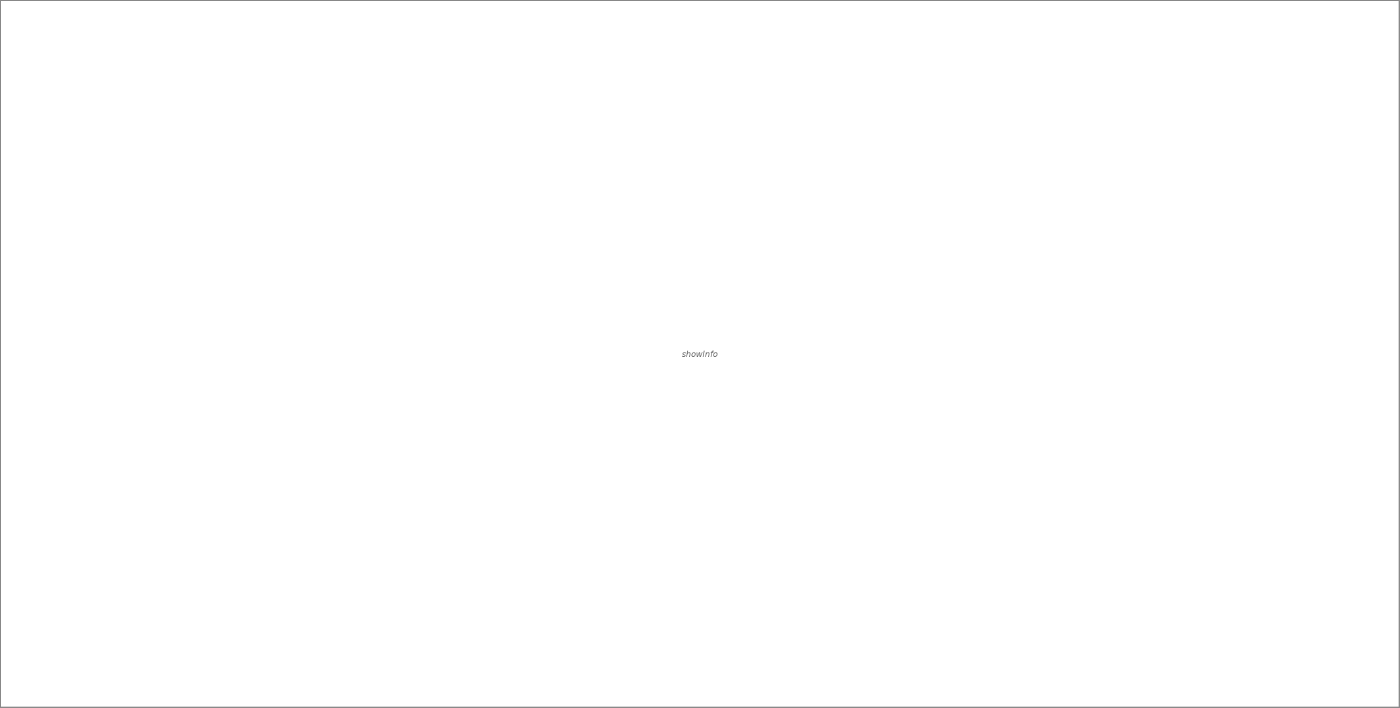
VISUALIZATION LogInf  // 1740x880
    TabControl (0,0 1740x880)
        shows showInfo(userData := gLog.HMIData)
        shows showInfo(userData := gDataChangeLog.HMIData)
        shows showInfo(userData := gDownTimeLog.HMIData)
        shows showInfo(userData := gBreakTimeLog.HMIData)
        shows showInfo(userData := gOperatorLog.HMIData)
        shows showInfo(userData := gRunningLog.HMIData)
        [1]: TabTitle=Data Change
        [2]: TabTitle=Error
        [3]: TabTitle=Time
        [4]: TabTitle=Operator
        [5]: TabTitle=Runing
END_VISUALIZATION

(* stored: Version 1.1.0.1, ProductVersion 3.1.4024.4
   Visu LogInf: Id {c207fd45-198c-419d-b43f-766d9dd09b38} *)
